{attribute 'qualified_only'}
VAR_GLOBAL
	// Füllstand (0-10V)
	Pegel:  INT;
END_VAR

(* stored: Version 1.1.0.1, ProductVersion 3.1.4024.5
   GVL AI: Id {10f5e73c-1377-4a8e-bddc-daf6fe97d7d3} *)
